// TIA Portal V18 export
FUNCTION_BLOCK "StopperCtrl"   // FB2600, LAD
TITLE = stopper program
{ S7_Optimized_Access := 'TRUE' }
// stored: AutoNumber false, MemoryReserve 100, SetENOAutomatically false
   VAR_INPUT
      i_SysRun : Bool;
      i_AutoMode : Bool;
      i_AutoRunnig : Bool;
      i_Reset : Bool;
      i_LineRunning : Bool;
      i_PalletArrivedNextStation : Bool;
      i_StopperSensor : Bool;   // local arrived sensor
      "i_Cyl-Home" : Bool;   // 顶升气缸原始位
      i_NextStationReady : Bool;
      i_PresentDelayTime : Time;
      i_ReleaseDelayTime : Time;
   END_VAR
   VAR_OUTPUT
      o_StopperClyWP : Bool;   // Stopper cylinder
      o_StopperClyHP : Bool;
   END_VAR
   VAR_IN_OUT
      io_NextyStopperStatus : Int;
      io_Interface : "UDT_StopperInterface";
      io_MotorCWRun : Bool;
      io_MotorCCWRun : Bool;
   END_VAR
   VAR RETAIN
      s_Sequence : Int;   // pulse flag
   END_VAR
   VAR
      s_SequenceEnable : Bool;
      s_SequenceFirstEnable : Bool;
      s_StopperSensorOnDelay { S7_SetPoint := 'True'} : TON_TIME;
      s_StopperSensorOffDelay { S7_SetPoint := 'True'} : TON_TIME;
      s_PalletMissingConfirmDelay { S7_SetPoint := 'True'} : TON_TIME;
      s_PalletToNextStationDelay { S7_SetPoint := 'True'} : TON_TIME;
      s_SequenceFirstAutoDelay { S7_SetPoint := 'True'} : TON_TIME;
      s_SequenceFirstAuto { S7_SetPoint := 'True'} : Int;
      s_StopperSensor : Bool;
      s_PalletArrivedNextStation : Bool;
      P : Array[0..10] of Bool;
   END_VAR
   VAR_TEMP
      t_AlwaysOn : Bool;
   END_VAR
   VAR_TEMP   // added for the SCL form of the ladder/FBD networks
      _w1 : Bool;
      _w2 : Bool;
      _w3 : Bool;
      _w4 : Bool;
   END_VAR
BEGIN

REGION Network 1: Always On
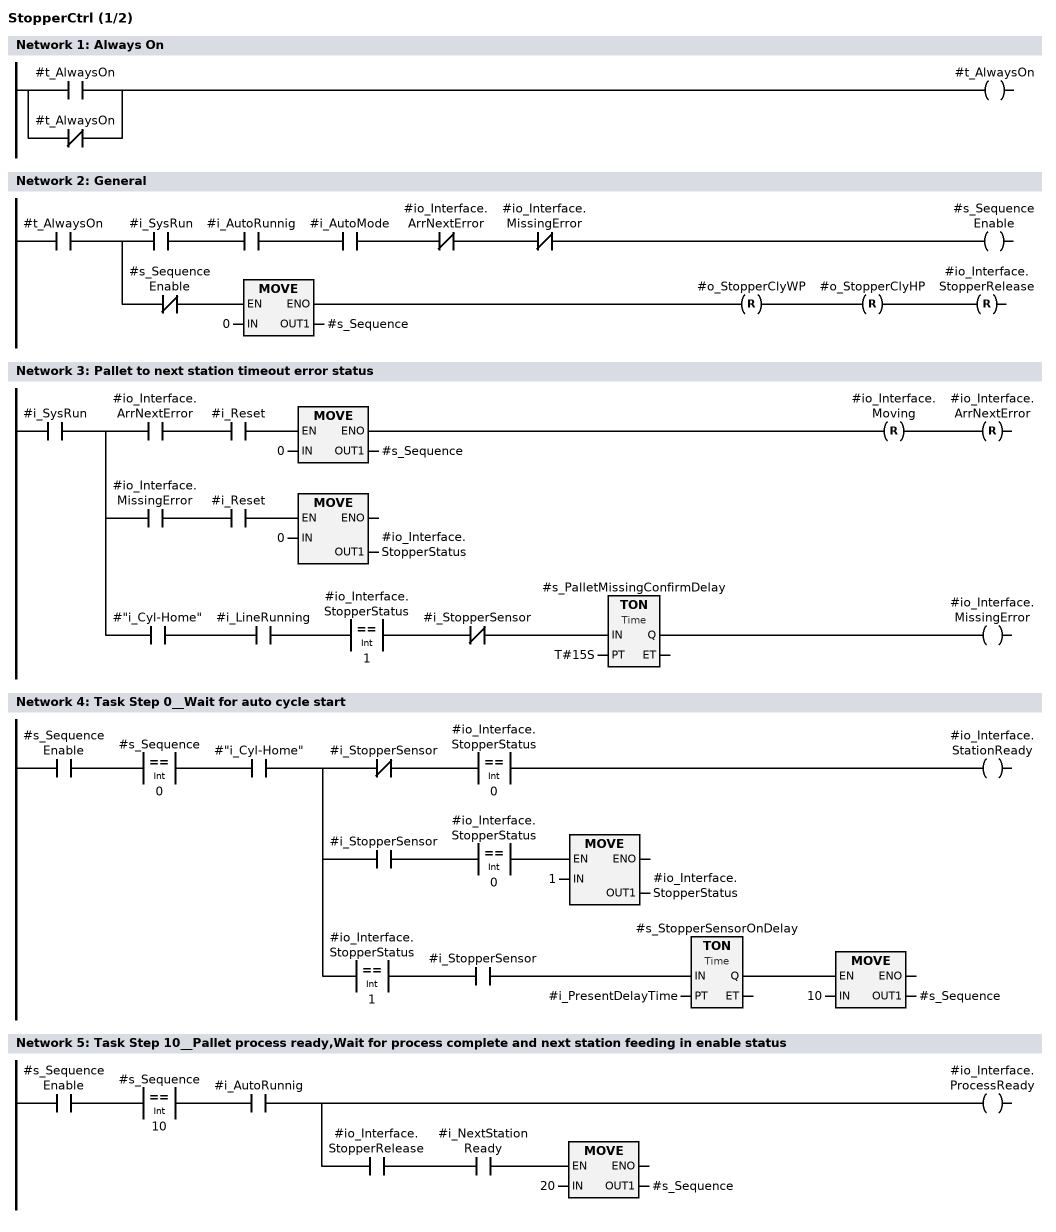
   RUNG wire#powerrail
      Contact( #t_AlwaysOn )
      wire#w1
      Coil( #t_AlwaysOn )
   END_RUNG
   RUNG wire#powerrail
      I_Contact( #t_AlwaysOn )
   END_RUNG wire#w1
   // the same network as SCL:
   #t_AlwaysOn := #t_AlwaysOn OR NOT #t_AlwaysOn;
END_REGION

REGION Network 2: General
   RUNG wire#powerrail
      Contact( #t_AlwaysOn )
      wire#w1
      Contact( #i_SysRun )
      Contact( #i_AutoRunnig )
      Contact( #i_AutoMode )
      I_Contact( #io_Interface.ArrNextError )
      I_Contact( #io_Interface.MissingError )
      Coil( #s_SequenceEnable )
   END_RUNG
   RUNG wire#w1
      I_Contact( #s_SequenceEnable )
      Move(in := 0, out1 => #s_Sequence)
      R_Coil( #o_StopperClyWP )
      R_Coil( #o_StopperClyHP )
      R_Coil( #io_Interface.StopperRelease )
   END_RUNG
   // the same network as SCL:
   #s_SequenceEnable := #t_AlwaysOn AND #i_SysRun AND #i_AutoRunnig AND #i_AutoMode AND NOT #io_Interface.ArrNextError AND NOT #io_Interface.MissingError;
   IF #t_AlwaysOn AND NOT #s_SequenceEnable THEN
       #s_Sequence := 0;
       #o_StopperClyWP := FALSE;
       #o_StopperClyHP := FALSE;
       #io_Interface.StopperRelease := FALSE;
   END_IF;
END_REGION

REGION Network 3: Pallet to next station timeout error status
   RUNG wire#powerrail
      Contact( #i_SysRun )
      wire#w1
      Contact( #io_Interface.ArrNextError )
      Contact( #i_Reset )
      Move(in := 0, out1 => #s_Sequence)
      R_Coil( #io_Interface.Moving )
      R_Coil( #io_Interface.ArrNextError )
   END_RUNG
   RUNG wire#w1
      Contact( #io_Interface.MissingError )
      Contact( #i_Reset )
      Move(in := 0, out1 => #io_Interface.StopperStatus)
   END_RUNG
   RUNG wire#w1
      Contact( #"i_Cyl-Home" )
      Contact( #i_LineRunning )
      { S7_Templates := "SrcType := Int" } EQ_Contact(in1 := #io_Interface.StopperStatus, in2 := 1)
      I_Contact( #i_StopperSensor )
      { S7_Templates := "time_type := Time" } #s_PalletMissingConfirmDelay.TON(pt := T#15S, et =>)
      Coil( #io_Interface.MissingError )
   END_RUNG
   // the same network as SCL:
   IF #i_SysRun AND #io_Interface.ArrNextError AND #i_Reset THEN
       #s_Sequence := 0;
       #io_Interface.Moving := FALSE;
       #io_Interface.ArrNextError := FALSE;
   END_IF;
   IF #i_SysRun AND #io_Interface.MissingError AND #i_Reset THEN #io_Interface.StopperStatus := 0; END_IF;
   #s_PalletMissingConfirmDelay(IN := #i_SysRun AND #"i_Cyl-Home" AND #i_LineRunning AND (#io_Interface.StopperStatus = 1) AND NOT #i_StopperSensor,   // TON
                           PT := T#15S);
   #io_Interface.MissingError := #s_PalletMissingConfirmDelay.Q;
END_REGION

REGION Network 4: Task Step 0__Wait for auto cycle start
   RUNG wire#powerrail
      Contact( #s_SequenceEnable )
      { S7_Templates := "SrcType := Int" } EQ_Contact(in1 := #s_Sequence, in2 := 0)
      Contact( #"i_Cyl-Home" )
      wire#w1
      I_Contact( #i_StopperSensor )
      { S7_Templates := "SrcType := Int" } EQ_Contact(in1 := #io_Interface.StopperStatus, in2 := 0)
      Coil( #io_Interface.StationReady )
   END_RUNG
   RUNG wire#w1
      Contact( #i_StopperSensor )
      { S7_Templates := "SrcType := Int" } EQ_Contact(in1 := #io_Interface.StopperStatus, in2 := 0)
      Move(in := 1, out1 => #io_Interface.StopperStatus)
   END_RUNG
   RUNG wire#w1
      { S7_Templates := "SrcType := Int" } EQ_Contact(in1 := #io_Interface.StopperStatus, in2 := 1)
      Contact( #i_StopperSensor )
      { S7_Templates := "time_type := Time" } #s_StopperSensorOnDelay.TON(pt := #i_PresentDelayTime, et =>)
      Move(in := 10, out1 => #s_Sequence)
   END_RUNG
   // the same network as SCL:
   #_w1 := #s_SequenceEnable AND (#s_Sequence = 0) AND #"i_Cyl-Home";
   #io_Interface.StationReady := #_w1 AND NOT #i_StopperSensor AND (#io_Interface.StopperStatus = 0);
   IF #_w1 AND #i_StopperSensor AND (#io_Interface.StopperStatus = 0) THEN
       #io_Interface.StopperStatus := 1;
   END_IF;
   #s_StopperSensorOnDelay(IN := #_w1 AND (#io_Interface.StopperStatus = 1) AND #i_StopperSensor,   // TON
                           PT := #i_PresentDelayTime);
   IF #s_StopperSensorOnDelay.Q THEN #s_Sequence := 10; END_IF;
END_REGION

REGION Network 5: Task Step 10__Pallet process ready,Wait for process complete and next station feeding in enable status
   RUNG wire#powerrail
      Contact( #s_SequenceEnable )
      { S7_Templates := "SrcType := Int" } EQ_Contact(in1 := #s_Sequence, in2 := 10)
      Contact( #i_AutoRunnig )
      wire#w1
      Coil( #io_Interface.ProcessReady )
   END_RUNG
   RUNG wire#w1
      Contact( #io_Interface.StopperRelease )
      Contact( #i_NextStationReady )
      Move(in := 20, out1 => #s_Sequence)
   END_RUNG
   // the same network as SCL:
   #io_Interface.ProcessReady := #s_SequenceEnable AND (#s_Sequence = 10) AND #i_AutoRunnig;
   IF #io_Interface.ProcessReady AND #io_Interface.StopperRelease AND #i_NextStationReady THEN
       #s_Sequence := 20;
   END_IF;
END_REGION

REGION Network 6: Task Step 20__Pallet releasing
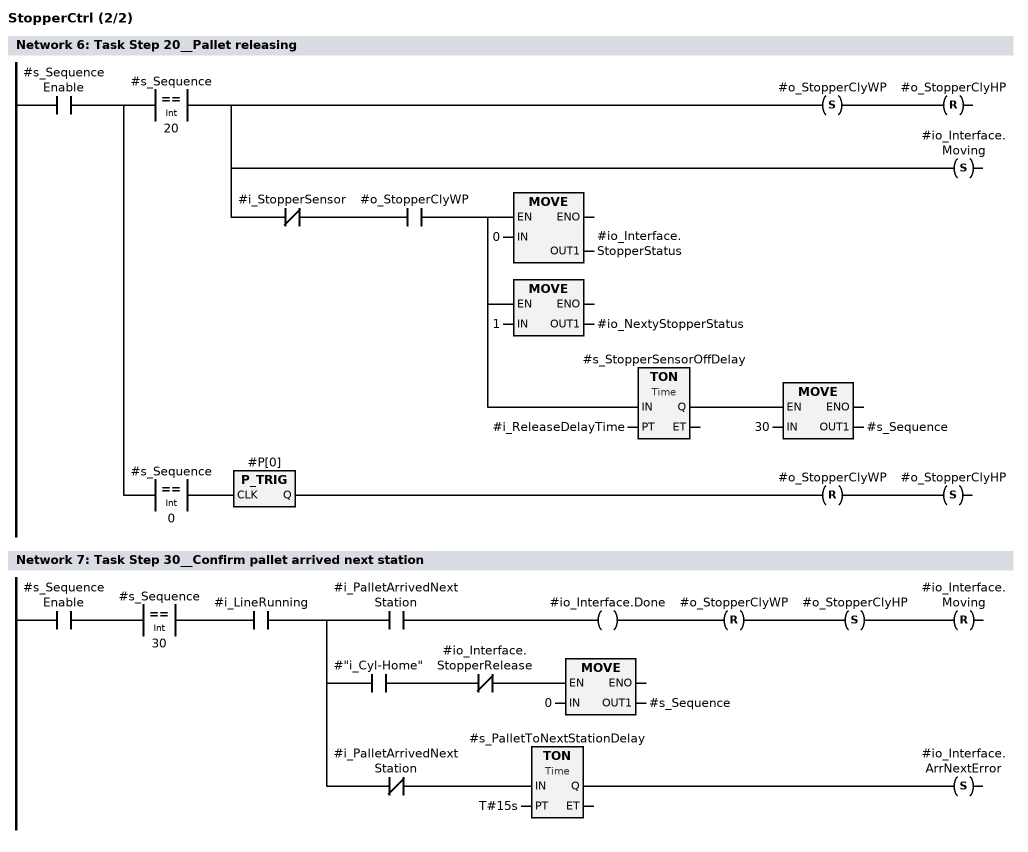
   RUNG wire#powerrail
      Contact( #s_SequenceEnable )
      wire#w1
      { S7_Templates := "SrcType := Int" } EQ_Contact(in1 := #s_Sequence, in2 := 20)
      wire#w2
      S_Coil( #o_StopperClyWP )
      R_Coil( #o_StopperClyHP )
   END_RUNG
   RUNG wire#w2
      S_Coil( #io_Interface.Moving )
   END_RUNG
   RUNG wire#w2
      I_Contact( #i_StopperSensor )
      Contact( #o_StopperClyWP )
      wire#w3
      Move(in := 0, out1 => #io_Interface.StopperStatus)
   END_RUNG
   RUNG wire#w3
      Move(in := 1, out1 => #io_NextyStopperStatus)
   END_RUNG
   RUNG wire#w3
      { S7_Templates := "time_type := Time" } #s_StopperSensorOffDelay.TON(pt := #i_ReleaseDelayTime, et =>)
      Move(in := 30, out1 => #s_Sequence)
   END_RUNG
   RUNG wire#w1
      { S7_Templates := "SrcType := Int" } EQ_Contact(in1 := #s_Sequence, in2 := 0)
      P_Trig( #P[0] )
      R_Coil( #o_StopperClyWP )
      S_Coil( #o_StopperClyHP )
   END_RUNG
   // the same network as SCL:
   #_w1 := #s_SequenceEnable AND (#s_Sequence = 20);
   IF #_w1 THEN
       #o_StopperClyWP := TRUE;
       #o_StopperClyHP := FALSE;
       #io_Interface.Moving := TRUE;
   END_IF;
   #_w2 := #_w1 AND NOT #i_StopperSensor AND #o_StopperClyWP;
   IF #_w2 THEN
       #io_Interface.StopperStatus := 0;
       #io_NextyStopperStatus := 1;
   END_IF;
   #s_StopperSensorOffDelay(IN := #_w2, PT := #i_ReleaseDelayTime);   // TON
   IF #s_StopperSensorOffDelay.Q THEN #s_Sequence := 30; END_IF;
   #_w3 := #s_SequenceEnable AND (#s_Sequence = 0);
   #_w4 := #_w3 AND NOT #P[0];   // rising edge
   #P[0] := #_w3;
   IF #_w4 THEN
       #o_StopperClyWP := FALSE;
       #o_StopperClyHP := TRUE;
   END_IF;
END_REGION

REGION Network 7: Task Step 30__Confirm pallet arrived next station
   RUNG wire#powerrail
      Contact( #s_SequenceEnable )
      { S7_Templates := "SrcType := Int" } EQ_Contact(in1 := #s_Sequence, in2 := 30)
      Contact( #i_LineRunning )
      wire#w1
      Contact( #i_PalletArrivedNextStation )
      Coil( #io_Interface.Done )
      R_Coil( #o_StopperClyWP )
      S_Coil( #o_StopperClyHP )
      R_Coil( #io_Interface.Moving )
   END_RUNG
   RUNG wire#w1
      Contact( #"i_Cyl-Home" )
      I_Contact( #io_Interface.StopperRelease )
      Move(in := 0, out1 => #s_Sequence)
   END_RUNG
   RUNG wire#w1
      I_Contact( #i_PalletArrivedNextStation )
      { S7_Templates := "time_type := Time" } #s_PalletToNextStationDelay.TON(pt := T#15s, et =>)
      S_Coil( #io_Interface.ArrNextError )
   END_RUNG
   // the same network as SCL:
   #_w1 := #s_SequenceEnable AND (#s_Sequence = 30) AND #i_LineRunning;
   #io_Interface.Done := #_w1 AND #i_PalletArrivedNextStation;
   IF #io_Interface.Done THEN
       #o_StopperClyWP := FALSE;
       #o_StopperClyHP := TRUE;
       #io_Interface.Moving := FALSE;
   END_IF;
   IF #_w1 AND #"i_Cyl-Home" AND NOT #io_Interface.StopperRelease THEN #s_Sequence := 0; END_IF;
   #s_PalletToNextStationDelay(IN := #_w1 AND NOT #i_PalletArrivedNextStation, PT := T#15s);   // TON
   IF #s_PalletToNextStationDelay.Q THEN #io_Interface.ArrNextError := TRUE; END_IF;
END_REGION
END_FUNCTION_BLOCK
